// TIA Portal V17 export
// export: Created 2021-12-03T08:12:56.2721734Z, ExportSetting WithDefaults, DisplayName Totally Integrated Automation Portal, DisplayVersion V17, DisplayName TIA Portal Openness, DisplayVersion V17, DisplayName TIA Portal Version Control Interface, DisplayVersion V17, DisplayName STEP 7 Professional, DisplayVersion V17, DisplayName STEP 7 Safety, DisplayVersion V17, DisplayName WinCC Advanced, DisplayVersion V17
DATA_BLOCK "GDB_DetLine"   // DB24
VERSION : 0.1
// stored: AutoNumber false, IsOnlyStoredInLoadMemory false, IsWriteProtectedInAS false
   VAR
      Request { ExternalVisible := 'False'; ExternalWritable := 'False'} : Struct   // External Input Structure
         DetLineStrtRq { ExternalVisible := 'False'; ExternalWritable := 'False'} : Bool;   // Detector Line: Start Request
         DetLineStpRq { ExternalVisible := 'False'; ExternalWritable := 'False'} : Bool;   // Detector Line: Stop Request
         DetLineSetRq { ExternalVisible := 'False'; ExternalWritable := 'False'} : Bool;   // Detector Line: Setup Request
         HiDoseMd { ExternalVisible := 'False'; ExternalWritable := 'False'} : Bool;   // High Dose Mode: 0=Off, 1=On
         VehMovDrct { ExternalVisible := 'False'; ExternalWritable := 'False'} : Bool;   // Vehicle Moving Direction: 0=Backward 1=Forward
         VehSpd { ExternalVisible := 'False'; ExternalWritable := 'False'} : Int;   // Vehicle Speed [m/min]
         ErgMd { ExternalVisible := 'False'; ExternalWritable := 'False'} : Int;   // Energie Mode
      END_STRUCT;
      Status { ExternalVisible := 'False'; ExternalWritable := 'False'} : Struct   // Детекторная линейка
         Con_Nok { ExternalVisible := 'False'; ExternalWritable := 'False'} : Bool;   // Connection Not Ok / 1=Нет соединения
         ConOk { ExternalVisible := 'False'; ExternalWritable := 'False'} : Bool;   // 1=Detector Line Connected / 1=Соединение Ок
         SyncStrt { ExternalVisible := 'False'; ExternalWritable := 'False'} : Bool;   // 1=Synchronizator Started / 1=Синхронизация запущена
         ScanAct { ExternalVisible := 'False'; ExternalWritable := 'False'} : Bool;   // 1=Scanning active / 1=Сканирование запущено
         RdyForScan { ExternalVisible := 'False'; ExternalWritable := 'False'} : Bool;   // 1=Ready for scanning / 1=Готов к сканированию
         State { ExternalVisible := 'False'; ExternalWritable := 'False'} : Int;   // State: 0=Error, 1=Service mode, 2=OK / Статус: 0=Ошибка, 1=Сервисный режим, 2=OK
         ErgMd { ExternalVisible := 'False'; ExternalWritable := 'False'} : Int;   // Energy Mode: 0=Reserved, 1=Low, 2=High, 3=Dual energy)
         TrigRate { ExternalVisible := 'False'; ExternalWritable := 'False'} : Int;   // Trigger Rate (Range 50-1000, Step 1)
         Error { ExternalVisible := 'False'; ExternalWritable := 'False'} : Bool;   // 1=Ошибка
         SrvsMd { ExternalVisible := 'False'; ExternalWritable := 'False'} : Bool;   // 1=Сервисный режим
         AutoMd { ExternalVisible := 'False'; ExternalWritable := 'False'} : Bool;   // 1=Ок
         EnrgMdLow { ExternalVisible := 'False'; ExternalWritable := 'False'} : Bool;
         EnrgMdHigh { ExternalVisible := 'False'; ExternalWritable := 'False'} : Bool;
         EnrgMdDual { ExternalVisible := 'False'; ExternalWritable := 'False'} : Bool;
      END_STRUCT;
   END_VAR
BEGIN
END_DATA_BLOCK
